PROGRAM PRG_FB_CSVDataExchanger_Test
VAR
	fbCSVDataExchanger	 		: FB_CSVDataExchanger;
	bFirstCycle 				: BOOL 		:= TRUE;
	
	sFileDir 					: STRING 	:= 'C:\TwinCAT\Tests\CSV_Reader\';
	sFileName 					: STRING 	:= 'Demo_Excel_File_FQC_Inputs_Test_2';
	sAmsNetId  					: STRING 	:= '';
	bAddHeader					: BOOL		:= FALSE;
	bCreateFile					: BOOL 		:= FALSE;
	bChangeSeparatorToComma		: BOOL 		:= FALSE;
	iMaxRowsNumber				: UDINT;
	iMaxColumnsNumber			: UDINT;
	
	bInit						: BOOL;
	bAbort						: BOOL;
	bReset						: BOOL;
	bSelectAll					: BOOL;
	bSelectRow					: BOOL;
	bSelectPath					: BOOL;
	bParseString				: BOOL;
			
	arrDatabase					: ARRAY[0..iMAX_CSV_ROWS - 1, 0..iMAX_CSV_COLUMNS - 1] OF STRING(iMAX_CSV_FIELD_LENGTH); (* Target PLC database *)	
	
	arrParsedString				: ARRAY[0..iMAX_CSV_COLUMNS - 1] OF STRING(iMAX_CSV_FIELD_LENGTH);	(* Target PLC database *)

	iColumnToSearch				: UDINT := 3;
	sValueToSearch			 	: WSTRING := "2";
	sRowResult				 	: STRING;
	
	
	iStateMachine				: USINT;
END_VAR

IF bFirstCycle THEN
	fbCSVDataExchanger.MR_FirstCycle(sFileDir 	:= sFileDir,
									sFileName 	:= sFileName,
									sAmsNetId 	:= '',
									bChangeSeparatorToComma := bChangeSeparatorToComma);									
	bFirstCycle := FALSE;
	
END_IF

IF bReset THEN
	bReset := FALSE;
	iStateMachine := 50;
	
ELSIF bAbort THEN
	bAbort := FALSE;
	iStateMachine := 60;

END_IF	

CASE iStateMachine OF
	0: 
		IF bInit THEN
			fbCSVDataExchanger.MR_Init();
			
			IF NOT fbCSVDataExchanger.Busy THEN
				bInit := FALSE;
				iStateMachine := 10;
				
			END_IF
		END_IF
		
	10: 
		IF bSelectAll THEN
			bSelectAll := FALSE;
			iStateMachine := 20;
		
		ELSIF bSelectRow THEN
			bSelectRow := FALSE;
			iStateMachine := 30;	

		ELSIF bSelectPath THEN
			bSelectPath := FALSE;
			iStateMachine := 40;	

		END_IF		
		
	20: 
		fbCSVDataExchanger.MR_SelectAll(iArrDataBaseAdr := ADR(arrDatabase));
		
		IF NOT fbCSVDataExchanger.Busy THEN
			iStateMachine := 10;
			
		END_IF
	
	30: 
		fbCSVDataExchanger.MR_SelectRow(iColumnToSearch := iColumnToSearch,
										sValueToSearch := WSTRING_TO_STRING(sValueToSearch),
										iArrParsedStringAdr := ADR(arrParsedString),
										sRowResult => sRowResult);
		
		IF NOT fbCSVDataExchanger.Busy THEN
			iStateMachine := 10;
			
		END_IF
	
	40:
		fbCSVDataExchanger.MR_SelectPath(sFileDir := sFileDir,
										sFileName := sFileName);
		
		IF NOT fbCSVDataExchanger.Busy THEN
			iStateMachine := 10;
			
		END_IF	

	50: 
		fbCSVDataExchanger.MR_Reset();
		
		IF NOT fbCSVDataExchanger.Busy THEN
			IF fbCSVDataExchanger.Active THEN
				iStateMachine := 10;
				
			ELSE
				iStateMachine := 0;
			
			END_IF
		END_IF
		
	60:
		fbCSVDataExchanger.MR_Abort();
	
		IF NOT fbCSVDataExchanger.Busy THEN
			iStateMachine := 0;
			
		END_IF
		
END_CASE

fbCSVDataExchanger();

END_PROGRAM

(* stored: Version 1.1.0.1, ProductVersion 3.1.4024.9
   POU PRG_FB_CSVDataExchanger_Test: Id {2f876af1-9d65-4ca4-80a8-394db43dc702}, SpecialFunc None *)
